// TIA Portal V19 export
TYPE "C106_VAR_IF_HSI_TYPIC"
   STRUCT
      BSC1 { ExternalAccessible := 'False'; ExternalVisible := 'False'; ExternalWritable := 'False'} : Bool;   // Hoogspanningsinstallatie beschikbaar
      BSC2 { ExternalAccessible := 'False'; ExternalVisible := 'False'; ExternalWritable := 'False'} : Bool;   // Hoogspanningsinstallatie niet beschikbaar
      BSC3 { ExternalAccessible := 'False'; ExternalVisible := 'False'; ExternalWritable := 'False'} : Bool;   // Hoogspanningsinstallatie beperkt beschikbaar
      WRE1 { ExternalAccessible := 'False'; ExternalVisible := 'False'; ExternalWritable := 'False'} : Bool;   // Werkingsregime: Netbedrijf
      WRE2 { ExternalAccessible := 'False'; ExternalVisible := 'False'; ExternalWritable := 'False'} : Bool;   // Werkingsregime: Parallelbedrijf
      WRE3 { ExternalAccessible := 'False'; ExternalVisible := 'False'; ExternalWritable := 'False'} : Bool;   // Werkingsregime: Eilandbedrijf
      LUS_TOE { ExternalAccessible := 'False'; ExternalVisible := 'False'; ExternalWritable := 'False'} : Bool;   // Hoogspanningslus is gesloten
      EXT_AUT { ExternalAccessible := 'False'; ExternalVisible := 'False'; ExternalWritable := 'False'} : Bool;   // Externe (hoofd) beveiliging aangesproken
      EXT_HW { ExternalAccessible := 'False'; ExternalVisible := 'False'; ExternalWritable := 'False'} : Bool;   // Sturings hardware (PLC) in storing
      STO { ExternalAccessible := 'False'; ExternalVisible := 'False'; ExternalWritable := 'False'} : Struct   // Opsomming van alle storingen
         A001 : Bool;   // Beveiliging aangesproken
         A002 : Bool;   // Hoogspanningsinstallatie in storing
         A003 : Bool;   // Algemene storing hoogspanningsinstallatie
         A004 : Bool;   // Hoogspanningslus is geopend
      END_STRUCT;
   END_STRUCT;
END_TYPE
